FUNCTION_BLOCK Necessidade_2_Equipamentos_ok_HMI (* Service Interface Function Block Type *)
  (* Standard: 61499-2 *)
  (* Version 0.0, 25/02/2026, template *)
  PACKAGE Hidryco.HidrycoLib;
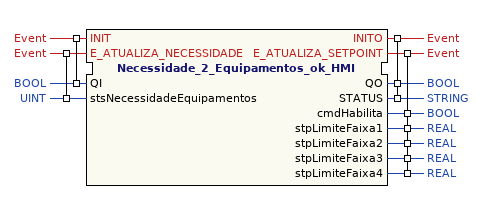
  EVENT_INPUT
    INIT WITH QI;
    E_ATUALIZA_NECESSIDADE WITH stsNecessidadeEquipamentos;
  END_EVENT
  EVENT_OUTPUT
    INITO WITH QO, STATUS;
    E_ATUALIZA_SETPOINT WITH stpLimiteFaixa1, stpLimiteFaixa2, stpLimiteFaixa3, stpLimiteFaixa4, cmdHabilita;
  END_EVENT
  VAR_INPUT
    QI : BOOL;
    stsNecessidadeEquipamentos : UINT;
  END_VAR
  VAR_OUTPUT
    QO : BOOL; (* Event Output Qualifier *)
    STATUS : STRING; (* Service Status *)
    cmdHabilita : BOOL;
    stpLimiteFaixa1 : REAL;
    stpLimiteFaixa2 : REAL;
    stpLimiteFaixa3 : REAL;
    stpLimiteFaixa4 : REAL;
  END_VAR
  SERVICE /
    SEQUENCE 
    END_SEQUENCE
  END_SERVICE
END_FUNCTION_BLOCK
